{attribute 'GeneratedUsingTerminal: EL2564-0000-0016'}
{attribute addProperty BoxType "EL2564-0000-0016"}
{attribute addProperty Id "StatusAT %I*Status_6BD97C373"}
{attribute addProperty CRC "810402373"}
{attribute addProperty Size "3"}
TYPE PWM_Inputs_Channel_304DC245 :
STRUCT
	{attribute addProperty Name "Status"}
	Status AT %I* : Status_6BD97C37;
END_STRUCT
END_TYPE

(* stored: Version 1.2.0.0, ProductVersion 3.1.4024.9
   DUT PWM_Inputs_Channel_304DC245: Id {4bde9691-483a-4be7-9b97-fbb4d34c1a02} *)
